{attribute 'qualified_only'}
VAR_GLOBAL
	Neutral:BOOL;
	Forward:BOOL;
	Reverse:BOOL;
	Button:BOOL;
	Raw:INT;
	Linear:INT;
	Cubic:INT;
END_VAR

(* stored: Version 1.1.0.1, ProductVersion 3.1.4024.0
   GVL Power_lever: Id {07f2c2bc-bf3d-4199-a09e-ef7fd167f7ad} *)
